(* IEC 61131-3 sources: CodesysTest/export/Function Blocks/Electric Solenoid/FB_ElectricSolenoid.pou, 1 file *)

(* ---- FB_ElectricSolenoid.pou.st ---- *)
(*#-#-#-#-#-#-#-#-#-#---Declaration---#-#-#-#-#-#-#-#-#-#-#-#-#*)

FUNCTION_BLOCK FB_ElectricSolenoid EXTENDS FB_BaseObject IMPLEMENTS ISimulateable, IUpDown
VAR_INPUT
	downFeedback : BOOL;
END_VAR
VAR_OUTPUT
	actuateSolenoid : BOOL;
END_VAR
VAR
	_simulateActive : BOOL;
END_VAR
(*#-#-#-#-#-#-#-#-#-#---Implementation---#-#-#-#-#-#-#-#-#-#-#-#-#*)
